FUNCTION ScaleRPS : RobotPoseSimple
VAR_INPUT
	c: 		LREAL;
	pose: 	RobotPoseSimple;
END_VAR
VAR
END_VAR

ScaleRPS.x		:= c*pose.x;	
ScaleRPS.y		:= c*pose.y;
ScaleRPS.theta	:= c*pose.theta;

END_FUNCTION

(* stored: Version 1.1.0.1, ProductVersion 3.1.4024.11
   POU ScaleRPS: Id {5a629f2e-08d7-4a8f-aed6-aac9109c3b54}, SpecialFunc None *)
